PROGRAM MAIN
VAR
	a:INT;
	b:INT;
	c:INT;
	add1:FB_ADD;
END_VAR

add1(in1:=a , in2:=b , out=>c );

END_PROGRAM

(* stored: Version 1.1.0.1, ProductVersion 3.1.4024.11
   POU MAIN: Id {851edad7-d12d-44ea-82ca-df7e8945d433}, SpecialFunc None *)
